// TIA Portal project "定时器模拟" (V15.1)

(* hardware
DEVICE "S7-1200 station_1"  S7-1200 Station
   slot 0: "Rack_0"  S7-1200 Rack  Rack  V1.0
   slot 1: "PLC_1"  CPU 1214C DC/DC/DC  6ES7 214-1AG40-0XB0  V4.2
*)

// ===== PLC "PLC_1"  CPU 1214C DC/DC/DC =====

VAR_GLOBAL   // PLC tag table "默认变量表"
   ""Tag_2"" AT %I1.0 : Bool;
   ""Tag_4"" AT %I1.1 : Bool;
   ""Tag_7"" AT %I1.3 : Bool;
   ""Tag_10"" AT %I1.2 : Bool;
   ""Tag_11"" AT %I1.4 : Bool;
   ""Tag_3"" AT %Q1.0 : Bool;
   ""Tag_6"" AT %Q1.1 : Bool;
   ""Tag_9"" AT %Q1.2 : Bool;
   ""Tag_13"" AT %Q1.3 : Bool;
END_VAR